FUNCTION Event_clear : BOOL
VAR_INPUT
END_VAR
VAR
	i: INT;
END_VAR

FOR i:=0 TO GVL.iAlarm_max DO
	GVL.events_alarm[i]	:= GVL.event_for_clear;
END_FOR

END_FUNCTION

(* stored: Version 1.1.0.1, ProductVersion 3.1.4024.12
   POU Event_clear: Id {72667ebe-a60a-4bd2-a00a-ed9dca273bf2}, SpecialFunc None *)
